// TIA Portal V18 export
FUNCTION "calc_speeds_from_mechanics" : Void   // FC15, FBD
{ S7_Optimized_Access := 'TRUE' }
VERSION : 0.1
// stored: AutoNumber true, IsIECCheckEnabled false, SetENOAutomatically false, UDAEnableTagReadback false
   VAR_INPUT
      mm_per_outputshaft_rev : Real;
      reduction_ration : Real;
      max_revs_at_10V : Real;
      counts_per_encoder_rev : Real;
      encoder_placed_on_motor : Bool;
   END_VAR
   VAR_OUTPUT
      dist_stop : Real;
      Vabsmax_mm_per_s : Real;
      counts_per_mm : Real;
      ER_params : Bool;
      er_w : WString;
   END_VAR
   VAR_IN_OUT
      para : "typeMotPara";
   END_VAR
   VAR_TEMP
      t_acceleration_s : Real;
      maxV_mm_per_min : Real;
      "a" : Real;
      v_abs_max : Real;
      dist_auto_done : Real;
      dist_absMax : Real;
      ER_param_1 : Bool;
      ER_param_2 : Bool;
      ER_param_3 : Bool;
      v_crawl : Real;
      t_mx : Real;
   END_VAR
   VAR CONSTANT
      erws1 : WString := WSTRING#'#t_acceleration_s = 0';
      erws2 : WString := WSTRING#'#v_abs_max = 0';
      erws3 : WString := WSTRING#'#t_mx =0';
   END_VAR
BEGIN

REGION Network 1 (SCL)

   #maxV_mm_per_min := #max_revs_at_10V / #reduction_ration * #mm_per_outputshaft_rev;

   #Vabsmax_mm_per_s := #maxV_mm_per_min / 60;
END_REGION

REGION Network 2 (SCL)
   IF #encoder_placed_on_motor THEN
       #counts_per_mm :=  #counts_per_encoder_rev * #reduction_ration / #mm_per_outputshaft_rev  ;
   ELSE
       #counts_per_mm := #counts_per_encoder_rev /  #mm_per_outputshaft_rev;

   END_IF;
END_REGION

REGION Network 4 (SCL)
   #v_crawl := #para.v_crawl_USER;

   #dist_stop:=#para.dist_stop_USER;
   #v_abs_max := #Vabsmax_mm_per_s;
   #para.v_absoluteMax_LOGIC := #v_abs_max;

   #t_mx := #t_acceleration_s := #para.t_acc_50Hz_USER;//:= #t_acc_50Hz_USER;
END_REGION

REGION Network 5 (SCL)
   #er_w := WSTRING#'no er';
   #ER_param_1 := #t_acceleration_s = 0;

   IF #ER_param_1 THEN
       #er_w := #erws1;
   END_IF;


   #ER_param_2 := #v_abs_max = 0;
   IF #ER_param_2 THEN
       #er_w := #erws2;
   END_IF;





   #ER_params := #ER_param_1 OR #ER_param_2 OR #ER_param_3;
END_REGION

REGION Network 6 (SCL)

   IF NOT #ER_params THEN
       #a := (#v_abs_max - #v_crawl) / #t_mx;
       #dist_absMax := #a * #t_mx * #t_mx / 2 + #v_crawl * #t_mx;
   ELSE
       #a := 0;
       #dist_absMax := 999;
   END_IF;
END_REGION

REGION Network 8 (SCL)

   #dist_auto_done := #dist_stop * 3;


   #para.dist_absMax_LOGIC := #dist_absMax;
   #para.dist_auto_done_LOGIC := #dist_auto_done;
   #para.v_auto_USER := LIMIT(MN := 0.0, IN := #para.v_auto_USER, MX := #v_abs_max);
   #para.v_manual_USER := LIMIT(MN := 0.0, IN := #para.v_manual_USER, MX := #v_abs_max);
END_REGION
END_FUNCTION
